FUNCTION_BLOCK FB_ProportionairRegulator
VAR_INPUT
END_VAR
VAR_OUTPUT
END_VAR
VAR_IN_OUT
	iq_stRegProp	:	ST_Proportionair;
END_VAR
VAR
END_VAR

(* A. Wallace 2015-10-7
Proportionair regulator control *)

(* Pressure signal conversion, max pressure out 1000 (I think...) *)
iq_stRegProp.iPressure := REAL_TO_INT(1000 * (INT_TO_REAL(iq_stRegProp.iPressureRaw) / 32767));

iq_stRegProp.iSetpoint := LIMIT(iq_stRegProp.iLoLimit, iq_stRegProp.iSetpoint, iq_stRegProp.iHiLimit);

iq_stRegProp.iSetpointRaw := REAL_TO_INT( (INT_TO_REAL(iq_stRegProp.iSetpoint)/1000)*32767);

END_FUNCTION_BLOCK

(* stored: Version 1.1.0.1, ProductVersion 3.1.0.26
   POU FB_ProportionairRegulator: Id {8353dc22-d596-4ee5-8fe9-fb2eb72364f8} *)
